FUNCTION_BLOCK FB_ListenerTest
VAR_INPUT
END_VAR
VAR_OUTPUT
END_VAR
VAR
	hr : HRESULT;
	
	bSubscribe : BOOL := TRUE;
	bSubscribed : BOOL;
	bUnSubscribe : BOOL;
	
	fbListenerFilter : FB_TcEventFilter; 
	fbMessageListener : FB_SampleListener;
END_VAR

fbMessageListener.Execute(); // retrieve messages and its texts


IF bSubscribe THEN 
	bSubscribe := FALSE;
	fbListenerFilter.Clear().EventClass.EqualTo(TC_EVENTS.PublisherEventClass.Message.uuidEventClass); //define all events (messages and alarms) from this eventclass   
	hr := fbMessageListener.Subscribe2(fbListenerFilter); //subscribe to retrieve defined events
	bSubscribed := fbMessageListener.bSubscribed;

END_IF 

IF bUnSubscribe THEN 
	bUnSubscribe := FALSE;
	hr := fbMessageListener.Unsubscribe();
	bSubscribed := fbMessageListener.bSubscribed;

END_IF

END_FUNCTION_BLOCK

(* stored: Version 1.1.0.1, ProductVersion 3.1.4024.12
   POU FB_ListenerTest: Id {3f56ea05-5d12-4cf3-aa32-b1078ff3baf8}, SpecialFunc None *)
